// TIA Portal V20 export
FUNCTION "CallManualOperationLines_EM" : Void   // FC66, LAD
// stored: SetENOAutomatically false
   VAR_INPUT
      disableUnit : Bool;
   END_VAR
   VAR_IN_OUT
      manualOperationEm : "LAF_typeManEm";
      manualOperationEmArea : Array[*] of "LAF_typeManOperationArea";
      manualOperationCms : Array[*] of "LAF_typeManOperation";
      Axis : Array[*] of "LBC_typeAxisControlInterface";
      Axis64Pos : Array[*] of "LBC_typeAxis64PosInterface";
      AxisSfotCam : Array[*] of "LER_typeSoftCamRelation";
      Sina : Array[*] of "LBC_typeSinaSpeedInterface";
      twoWayAcutor : Array[*] of "LBC_typeTwoWayActuatorInterface";
      Status : Array[*] of Word;
      errorID : Array[*] of Word;
   END_VAR
   VAR_TEMP
      tempLowerBoundAxis : Int;
      tempUpperBoundAxis : Int;
      tempLowerBoundAxis64Pos : Int;
      tempUpperBoundAxis64Pos : Int;
      tempLowerBoundSina : Int;
      tempUpperBoundSina : Int;
      tempLowerBoundTwoWayAct : Int;
      tempUpperBoundTwoWayAct : Int;
      tempEnd : Bool;
   END_VAR
BEGIN

REGION Network 1: Detect lower and upper bound of the array for further processing
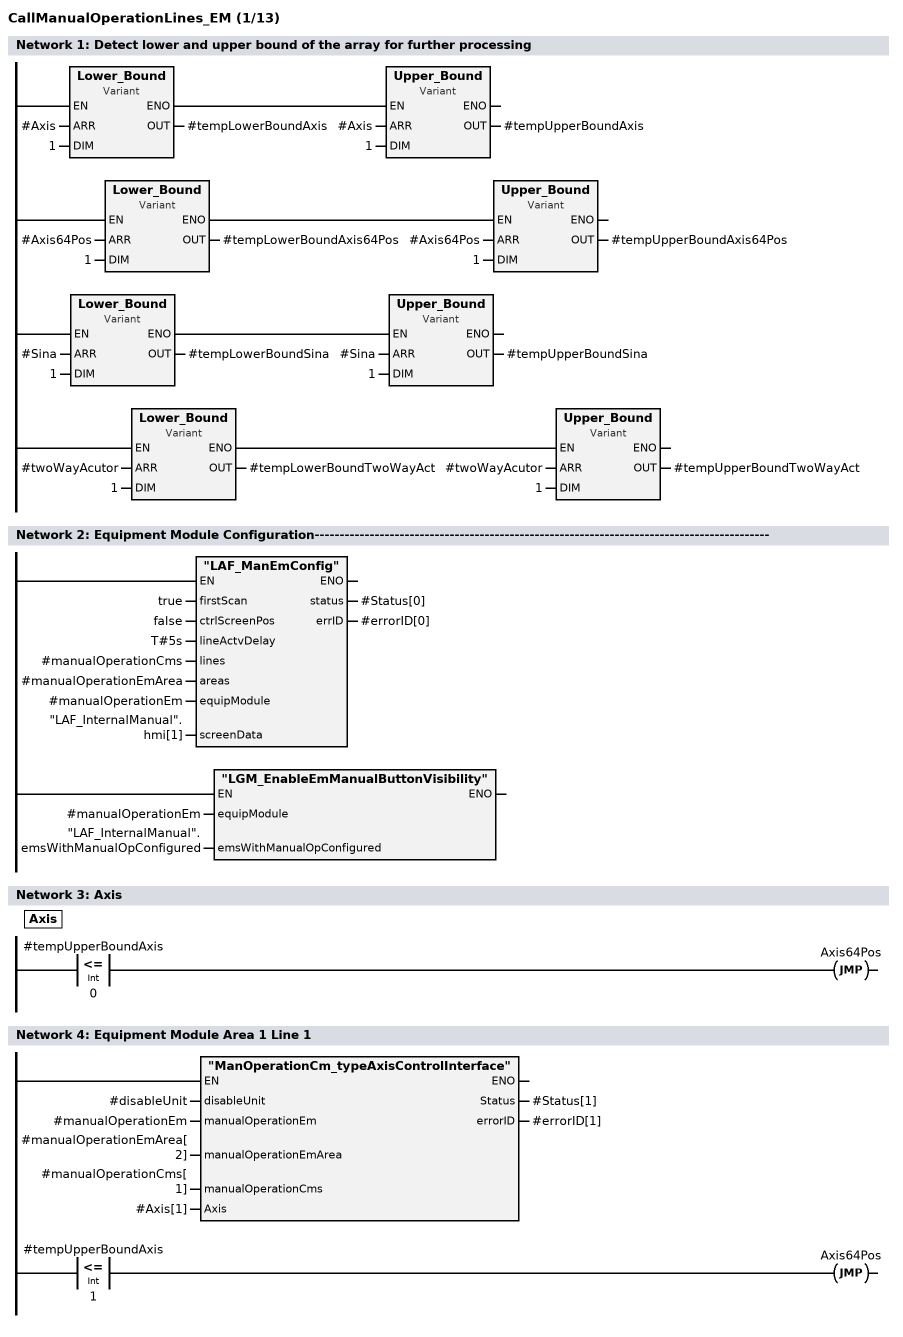
   // no SCL statement known for Lower_Bound, Upper_Bound: written as a call
   // ENO of a box is taken as its EN; it also drops when the box reports an error
   Lower_Bound(arr := #Axis, dim := 1, out => #tempLowerBoundAxis);
   Upper_Bound(arr := #Axis, dim := 1, out => #tempUpperBoundAxis);
   Lower_Bound(arr := #Axis64Pos, dim := 1, out => #tempLowerBoundAxis64Pos);
   Upper_Bound(arr := #Axis64Pos, dim := 1, out => #tempUpperBoundAxis64Pos);
   Lower_Bound(arr := #Sina, dim := 1, out => #tempLowerBoundSina);
   Upper_Bound(arr := #Sina, dim := 1, out => #tempUpperBoundSina);
   Lower_Bound(arr := #twoWayAcutor, dim := 1, out => #tempLowerBoundTwoWayAct);
   Upper_Bound(arr := #twoWayAcutor, dim := 1, out => #tempUpperBoundTwoWayAct);
END_REGION

REGION Network 2: Equipment Module Configuration-------------------------------------------------------------------------------------------
   RUNG wire#powerrail
      "LAF_ManEmConfig"(firstScan := true, ctrlScreenPos := false, lineActvDelay := T#5s, lines := #manualOperationCms, areas := #manualOperationEmArea, equipModule := #manualOperationEm, screenData := "LAF_InternalManual".hmi[1], status => #Status[0], errID => #errorID[0])
   END_RUNG
   RUNG wire#powerrail
      "LGM_EnableEmManualButtonVisibility"(equipModule := #manualOperationEm, emsWithManualOpConfigured := "LAF_InternalManual".emsWithManualOpConfigured)
   END_RUNG
   // the same network as SCL:
   "LAF_ManEmConfig"(firstScan := true,
                     ctrlScreenPos := false,
                     lineActvDelay := T#5s,
                     lines := #manualOperationCms,
                     areas := #manualOperationEmArea,
                     equipModule := #manualOperationEm,
                     screenData := "LAF_InternalManual".hmi[1],
                     status => #Status[0],
                     errID => #errorID[0]);
   "LGM_EnableEmManualButtonVisibility"(equipModule := #manualOperationEm,
                           emsWithManualOpConfigured := "LAF_InternalManual".emsWithManualOpConfigured);
END_REGION

REGION Network 3: Axis
   Label( Axis )
   RUNG wire#powerrail
      { S7_Templates := "SrcType := Int" } LE_Contact(in1 := #tempUpperBoundAxis, in2 := 0)
      JumpCoil( Axis64Pos )
   END_RUNG
   // the same network as SCL:
   Axis:
   IF #tempUpperBoundAxis <= 0 THEN GOTO Axis64Pos; END_IF;
END_REGION

REGION Network 4: Equipment Module Area 1 Line 1
   RUNG wire#powerrail
      "ManOperationCm_typeAxisControlInterface"(disableUnit := #disableUnit, manualOperationEm := #manualOperationEm, manualOperationEmArea := #manualOperationEmArea[2], manualOperationCms := #manualOperationCms[1], Axis := #Axis[1], Status => #Status[1], errorID => #errorID[1])
   END_RUNG
   RUNG wire#powerrail
      { S7_Templates := "SrcType := Int" } LE_Contact(in1 := #tempUpperBoundAxis, in2 := 1)
      JumpCoil( Axis64Pos )
   END_RUNG
   // the same network as SCL:
   "ManOperationCm_typeAxisControlInterface"(disableUnit := #disableUnit,
                           manualOperationEm := #manualOperationEm,
                           manualOperationEmArea := #manualOperationEmArea[2],
                           manualOperationCms := #manualOperationCms[1],
                           Axis := #Axis[1],
                           Status => #Status[1],
                           errorID => #errorID[1]);
   IF #tempUpperBoundAxis <= 1 THEN GOTO Axis64Pos; END_IF;
END_REGION

REGION Network 5: Equipment Module Area 1 Line 2
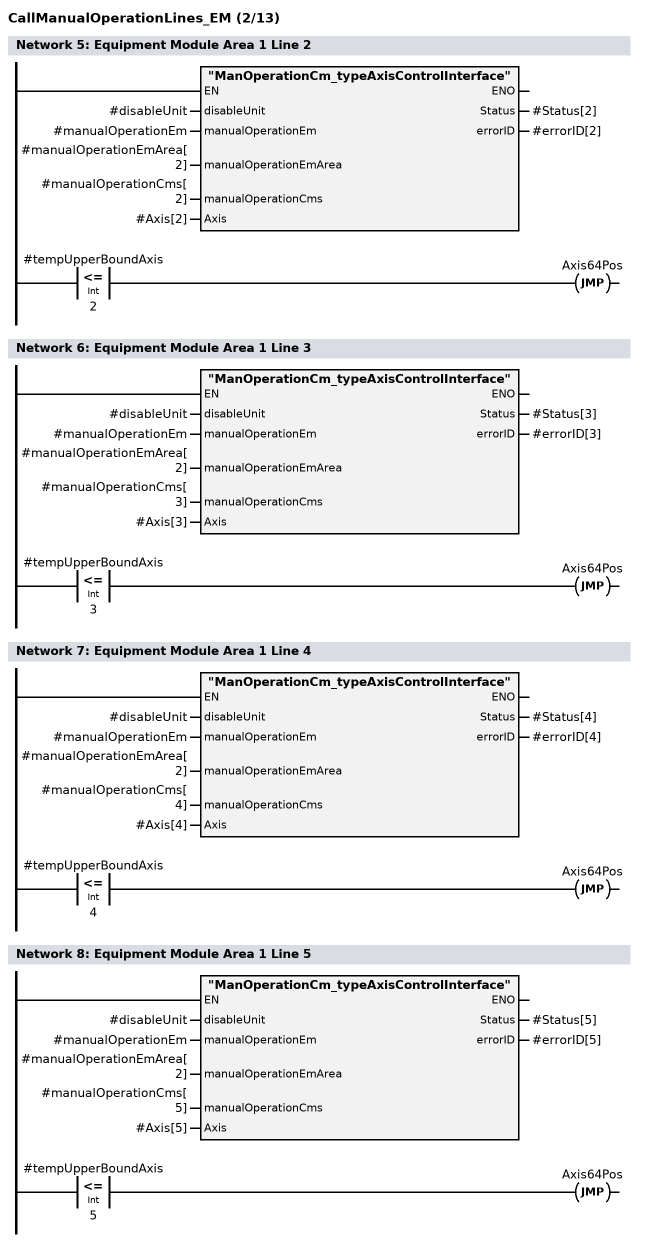
   RUNG wire#powerrail
      "ManOperationCm_typeAxisControlInterface"(disableUnit := #disableUnit, manualOperationEm := #manualOperationEm, manualOperationEmArea := #manualOperationEmArea[2], manualOperationCms := #manualOperationCms[2], Axis := #Axis[2], Status => #Status[2], errorID => #errorID[2])
   END_RUNG
   RUNG wire#powerrail
      { S7_Templates := "SrcType := Int" } LE_Contact(in1 := #tempUpperBoundAxis, in2 := 2)
      JumpCoil( Axis64Pos )
   END_RUNG
   // the same network as SCL:
   "ManOperationCm_typeAxisControlInterface"(disableUnit := #disableUnit,
                           manualOperationEm := #manualOperationEm,
                           manualOperationEmArea := #manualOperationEmArea[2],
                           manualOperationCms := #manualOperationCms[2],
                           Axis := #Axis[2],
                           Status => #Status[2],
                           errorID => #errorID[2]);
   IF #tempUpperBoundAxis <= 2 THEN GOTO Axis64Pos; END_IF;
END_REGION

REGION Network 6: Equipment Module Area 1 Line 3
   RUNG wire#powerrail
      "ManOperationCm_typeAxisControlInterface"(disableUnit := #disableUnit, manualOperationEm := #manualOperationEm, manualOperationEmArea := #manualOperationEmArea[2], manualOperationCms := #manualOperationCms[3], Axis := #Axis[3], Status => #Status[3], errorID => #errorID[3])
   END_RUNG
   RUNG wire#powerrail
      { S7_Templates := "SrcType := Int" } LE_Contact(in1 := #tempUpperBoundAxis, in2 := 3)
      JumpCoil( Axis64Pos )
   END_RUNG
   // the same network as SCL:
   "ManOperationCm_typeAxisControlInterface"(disableUnit := #disableUnit,
                           manualOperationEm := #manualOperationEm,
                           manualOperationEmArea := #manualOperationEmArea[2],
                           manualOperationCms := #manualOperationCms[3],
                           Axis := #Axis[3],
                           Status => #Status[3],
                           errorID => #errorID[3]);
   IF #tempUpperBoundAxis <= 3 THEN GOTO Axis64Pos; END_IF;
END_REGION

REGION Network 7: Equipment Module Area 1 Line 4
   RUNG wire#powerrail
      "ManOperationCm_typeAxisControlInterface"(disableUnit := #disableUnit, manualOperationEm := #manualOperationEm, manualOperationEmArea := #manualOperationEmArea[2], manualOperationCms := #manualOperationCms[4], Axis := #Axis[4], Status => #Status[4], errorID => #errorID[4])
   END_RUNG
   RUNG wire#powerrail
      { S7_Templates := "SrcType := Int" } LE_Contact(in1 := #tempUpperBoundAxis, in2 := 4)
      JumpCoil( Axis64Pos )
   END_RUNG
   // the same network as SCL:
   "ManOperationCm_typeAxisControlInterface"(disableUnit := #disableUnit,
                           manualOperationEm := #manualOperationEm,
                           manualOperationEmArea := #manualOperationEmArea[2],
                           manualOperationCms := #manualOperationCms[4],
                           Axis := #Axis[4],
                           Status => #Status[4],
                           errorID => #errorID[4]);
   IF #tempUpperBoundAxis <= 4 THEN GOTO Axis64Pos; END_IF;
END_REGION

REGION Network 8: Equipment Module Area 1 Line 5
   RUNG wire#powerrail
      "ManOperationCm_typeAxisControlInterface"(disableUnit := #disableUnit, manualOperationEm := #manualOperationEm, manualOperationEmArea := #manualOperationEmArea[2], manualOperationCms := #manualOperationCms[5], Axis := #Axis[5], Status => #Status[5], errorID => #errorID[5])
   END_RUNG
   RUNG wire#powerrail
      { S7_Templates := "SrcType := Int" } LE_Contact(in1 := #tempUpperBoundAxis, in2 := 5)
      JumpCoil( Axis64Pos )
   END_RUNG
   // the same network as SCL:
   "ManOperationCm_typeAxisControlInterface"(disableUnit := #disableUnit,
                           manualOperationEm := #manualOperationEm,
                           manualOperationEmArea := #manualOperationEmArea[2],
                           manualOperationCms := #manualOperationCms[5],
                           Axis := #Axis[5],
                           Status => #Status[5],
                           errorID => #errorID[5]);
   IF #tempUpperBoundAxis <= 5 THEN GOTO Axis64Pos; END_IF;
END_REGION

REGION Network 9: Equipment Module Area 1 Line 6
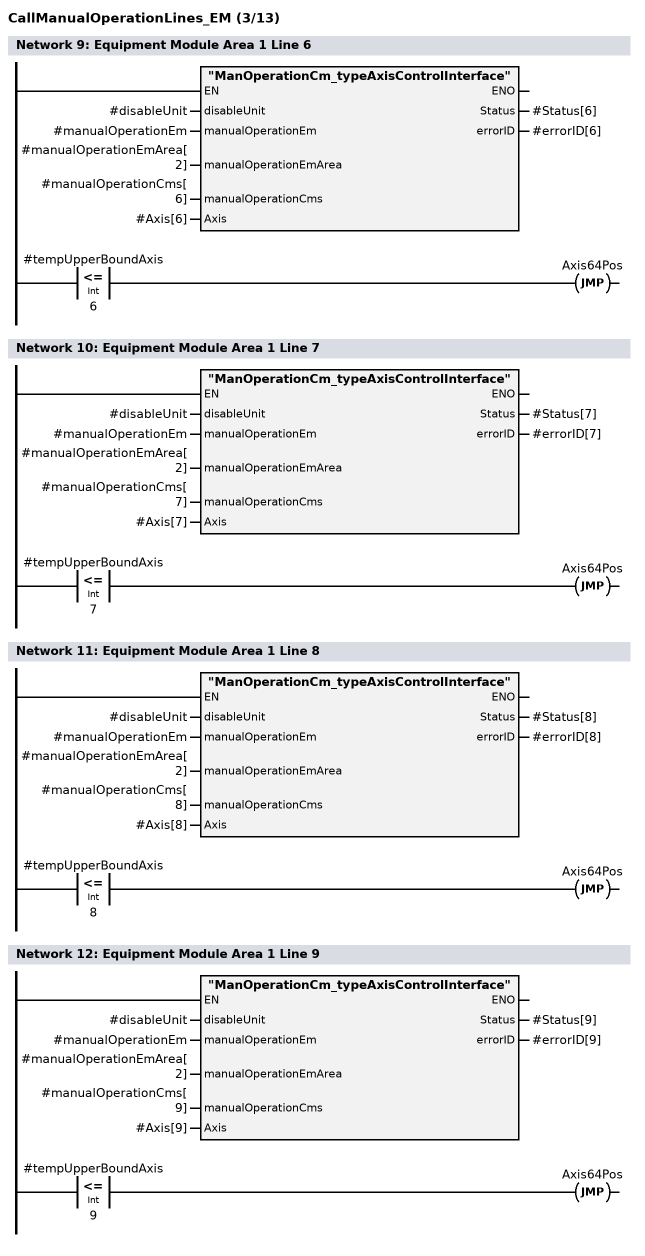
   RUNG wire#powerrail
      "ManOperationCm_typeAxisControlInterface"(disableUnit := #disableUnit, manualOperationEm := #manualOperationEm, manualOperationEmArea := #manualOperationEmArea[2], manualOperationCms := #manualOperationCms[6], Axis := #Axis[6], Status => #Status[6], errorID => #errorID[6])
   END_RUNG
   RUNG wire#powerrail
      { S7_Templates := "SrcType := Int" } LE_Contact(in1 := #tempUpperBoundAxis, in2 := 6)
      JumpCoil( Axis64Pos )
   END_RUNG
   // the same network as SCL:
   "ManOperationCm_typeAxisControlInterface"(disableUnit := #disableUnit,
                           manualOperationEm := #manualOperationEm,
                           manualOperationEmArea := #manualOperationEmArea[2],
                           manualOperationCms := #manualOperationCms[6],
                           Axis := #Axis[6],
                           Status => #Status[6],
                           errorID => #errorID[6]);
   IF #tempUpperBoundAxis <= 6 THEN GOTO Axis64Pos; END_IF;
END_REGION

REGION Network 10: Equipment Module Area 1 Line 7
   RUNG wire#powerrail
      "ManOperationCm_typeAxisControlInterface"(disableUnit := #disableUnit, manualOperationEm := #manualOperationEm, manualOperationEmArea := #manualOperationEmArea[2], manualOperationCms := #manualOperationCms[7], Axis := #Axis[7], Status => #Status[7], errorID => #errorID[7])
   END_RUNG
   RUNG wire#powerrail
      { S7_Templates := "SrcType := Int" } LE_Contact(in1 := #tempUpperBoundAxis, in2 := 7)
      JumpCoil( Axis64Pos )
   END_RUNG
   // the same network as SCL:
   "ManOperationCm_typeAxisControlInterface"(disableUnit := #disableUnit,
                           manualOperationEm := #manualOperationEm,
                           manualOperationEmArea := #manualOperationEmArea[2],
                           manualOperationCms := #manualOperationCms[7],
                           Axis := #Axis[7],
                           Status => #Status[7],
                           errorID => #errorID[7]);
   IF #tempUpperBoundAxis <= 7 THEN GOTO Axis64Pos; END_IF;
END_REGION

REGION Network 11: Equipment Module Area 1 Line 8
   RUNG wire#powerrail
      "ManOperationCm_typeAxisControlInterface"(disableUnit := #disableUnit, manualOperationEm := #manualOperationEm, manualOperationEmArea := #manualOperationEmArea[2], manualOperationCms := #manualOperationCms[8], Axis := #Axis[8], Status => #Status[8], errorID => #errorID[8])
   END_RUNG
   RUNG wire#powerrail
      { S7_Templates := "SrcType := Int" } LE_Contact(in1 := #tempUpperBoundAxis, in2 := 8)
      JumpCoil( Axis64Pos )
   END_RUNG
   // the same network as SCL:
   "ManOperationCm_typeAxisControlInterface"(disableUnit := #disableUnit,
                           manualOperationEm := #manualOperationEm,
                           manualOperationEmArea := #manualOperationEmArea[2],
                           manualOperationCms := #manualOperationCms[8],
                           Axis := #Axis[8],
                           Status => #Status[8],
                           errorID => #errorID[8]);
   IF #tempUpperBoundAxis <= 8 THEN GOTO Axis64Pos; END_IF;
END_REGION

REGION Network 12: Equipment Module Area 1 Line 9
   RUNG wire#powerrail
      "ManOperationCm_typeAxisControlInterface"(disableUnit := #disableUnit, manualOperationEm := #manualOperationEm, manualOperationEmArea := #manualOperationEmArea[2], manualOperationCms := #manualOperationCms[9], Axis := #Axis[9], Status => #Status[9], errorID => #errorID[9])
   END_RUNG
   RUNG wire#powerrail
      { S7_Templates := "SrcType := Int" } LE_Contact(in1 := #tempUpperBoundAxis, in2 := 9)
      JumpCoil( Axis64Pos )
   END_RUNG
   // the same network as SCL:
   "ManOperationCm_typeAxisControlInterface"(disableUnit := #disableUnit,
                           manualOperationEm := #manualOperationEm,
                           manualOperationEmArea := #manualOperationEmArea[2],
                           manualOperationCms := #manualOperationCms[9],
                           Axis := #Axis[9],
                           Status => #Status[9],
                           errorID => #errorID[9]);
   IF #tempUpperBoundAxis <= 9 THEN GOTO Axis64Pos; END_IF;
END_REGION

REGION Network 13: Equipment Module Area 1 Line 10
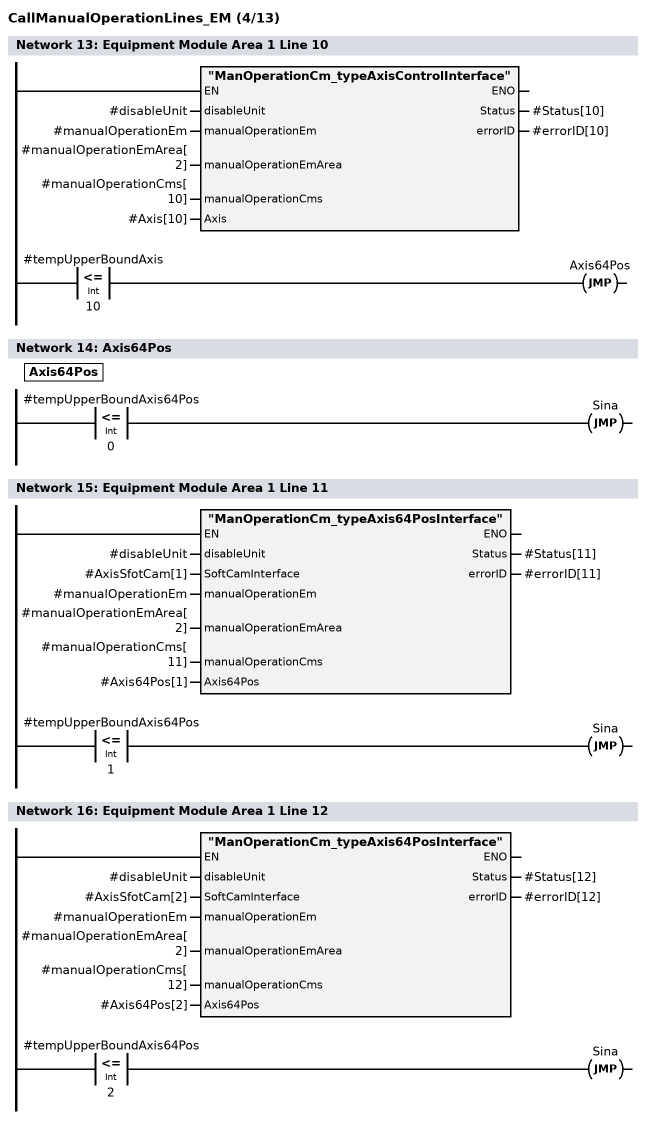
   RUNG wire#powerrail
      "ManOperationCm_typeAxisControlInterface"(disableUnit := #disableUnit, manualOperationEm := #manualOperationEm, manualOperationEmArea := #manualOperationEmArea[2], manualOperationCms := #manualOperationCms[10], Axis := #Axis[10], Status => #Status[10], errorID => #errorID[10])
   END_RUNG
   RUNG wire#powerrail
      { S7_Templates := "SrcType := Int" } LE_Contact(in1 := #tempUpperBoundAxis, in2 := 10)
      JumpCoil( Axis64Pos )
   END_RUNG
   // the same network as SCL:
   "ManOperationCm_typeAxisControlInterface"(disableUnit := #disableUnit,
                           manualOperationEm := #manualOperationEm,
                           manualOperationEmArea := #manualOperationEmArea[2],
                           manualOperationCms := #manualOperationCms[10],
                           Axis := #Axis[10],
                           Status => #Status[10],
                           errorID => #errorID[10]);
   IF #tempUpperBoundAxis <= 10 THEN GOTO Axis64Pos; END_IF;
END_REGION

REGION Network 14: Axis64Pos
   Label( Axis64Pos )
   RUNG wire#powerrail
      { S7_Templates := "SrcType := Int" } LE_Contact(in1 := #tempUpperBoundAxis64Pos, in2 := 0)
      JumpCoil( Sina )
   END_RUNG
   // the same network as SCL:
   Axis64Pos:
   IF #tempUpperBoundAxis64Pos <= 0 THEN GOTO Sina; END_IF;
END_REGION

REGION Network 15: Equipment Module Area 1 Line 11
   RUNG wire#powerrail
      "ManOperationCm_typeAxis64PosInterface"(disableUnit := #disableUnit, SoftCamInterface := #AxisSfotCam[1], manualOperationEm := #manualOperationEm, manualOperationEmArea := #manualOperationEmArea[2], manualOperationCms := #manualOperationCms[11], Axis64Pos := #Axis64Pos[1], Status => #Status[11], errorID => #errorID[11])
   END_RUNG
   RUNG wire#powerrail
      { S7_Templates := "SrcType := Int" } LE_Contact(in1 := #tempUpperBoundAxis64Pos, in2 := 1)
      JumpCoil( Sina )
   END_RUNG
   // the same network as SCL:
   "ManOperationCm_typeAxis64PosInterface"(disableUnit := #disableUnit,
                           SoftCamInterface := #AxisSfotCam[1],
                           manualOperationEm := #manualOperationEm,
                           manualOperationEmArea := #manualOperationEmArea[2],
                           manualOperationCms := #manualOperationCms[11],
                           Axis64Pos := #Axis64Pos[1],
                           Status => #Status[11],
                           errorID => #errorID[11]);
   IF #tempUpperBoundAxis64Pos <= 1 THEN GOTO Sina; END_IF;
END_REGION

REGION Network 16: Equipment Module Area 1 Line 12
   RUNG wire#powerrail
      "ManOperationCm_typeAxis64PosInterface"(disableUnit := #disableUnit, SoftCamInterface := #AxisSfotCam[2], manualOperationEm := #manualOperationEm, manualOperationEmArea := #manualOperationEmArea[2], manualOperationCms := #manualOperationCms[12], Axis64Pos := #Axis64Pos[2], Status => #Status[12], errorID => #errorID[12])
   END_RUNG
   RUNG wire#powerrail
      { S7_Templates := "SrcType := Int" } LE_Contact(in1 := #tempUpperBoundAxis64Pos, in2 := 2)
      JumpCoil( Sina )
   END_RUNG
   // the same network as SCL:
   "ManOperationCm_typeAxis64PosInterface"(disableUnit := #disableUnit,
                           SoftCamInterface := #AxisSfotCam[2],
                           manualOperationEm := #manualOperationEm,
                           manualOperationEmArea := #manualOperationEmArea[2],
                           manualOperationCms := #manualOperationCms[12],
                           Axis64Pos := #Axis64Pos[2],
                           Status => #Status[12],
                           errorID => #errorID[12]);
   IF #tempUpperBoundAxis64Pos <= 2 THEN GOTO Sina; END_IF;
END_REGION

REGION Network 17: Equipment Module Area 1 Line 13
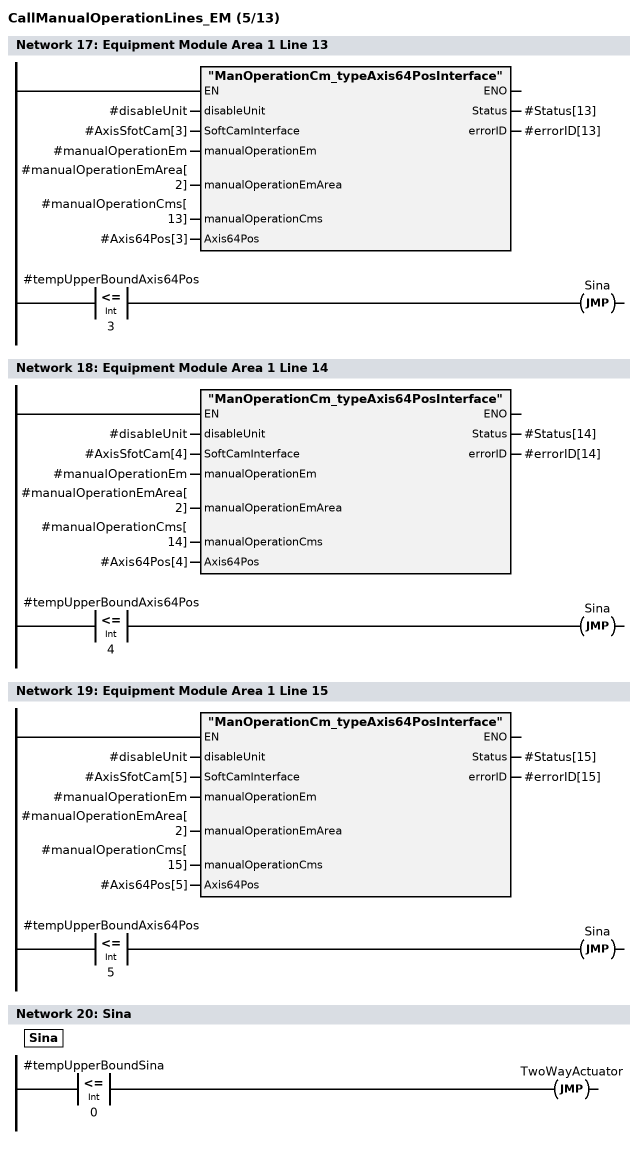
   RUNG wire#powerrail
      "ManOperationCm_typeAxis64PosInterface"(disableUnit := #disableUnit, SoftCamInterface := #AxisSfotCam[3], manualOperationEm := #manualOperationEm, manualOperationEmArea := #manualOperationEmArea[2], manualOperationCms := #manualOperationCms[13], Axis64Pos := #Axis64Pos[3], Status => #Status[13], errorID => #errorID[13])
   END_RUNG
   RUNG wire#powerrail
      { S7_Templates := "SrcType := Int" } LE_Contact(in1 := #tempUpperBoundAxis64Pos, in2 := 3)
      JumpCoil( Sina )
   END_RUNG
   // the same network as SCL:
   "ManOperationCm_typeAxis64PosInterface"(disableUnit := #disableUnit,
                           SoftCamInterface := #AxisSfotCam[3],
                           manualOperationEm := #manualOperationEm,
                           manualOperationEmArea := #manualOperationEmArea[2],
                           manualOperationCms := #manualOperationCms[13],
                           Axis64Pos := #Axis64Pos[3],
                           Status => #Status[13],
                           errorID => #errorID[13]);
   IF #tempUpperBoundAxis64Pos <= 3 THEN GOTO Sina; END_IF;
END_REGION

REGION Network 18: Equipment Module Area 1 Line 14
   RUNG wire#powerrail
      "ManOperationCm_typeAxis64PosInterface"(disableUnit := #disableUnit, SoftCamInterface := #AxisSfotCam[4], manualOperationEm := #manualOperationEm, manualOperationEmArea := #manualOperationEmArea[2], manualOperationCms := #manualOperationCms[14], Axis64Pos := #Axis64Pos[4], Status => #Status[14], errorID => #errorID[14])
   END_RUNG
   RUNG wire#powerrail
      { S7_Templates := "SrcType := Int" } LE_Contact(in1 := #tempUpperBoundAxis64Pos, in2 := 4)
      JumpCoil( Sina )
   END_RUNG
   // the same network as SCL:
   "ManOperationCm_typeAxis64PosInterface"(disableUnit := #disableUnit,
                           SoftCamInterface := #AxisSfotCam[4],
                           manualOperationEm := #manualOperationEm,
                           manualOperationEmArea := #manualOperationEmArea[2],
                           manualOperationCms := #manualOperationCms[14],
                           Axis64Pos := #Axis64Pos[4],
                           Status => #Status[14],
                           errorID => #errorID[14]);
   IF #tempUpperBoundAxis64Pos <= 4 THEN GOTO Sina; END_IF;
END_REGION

REGION Network 19: Equipment Module Area 1 Line 15
   RUNG wire#powerrail
      "ManOperationCm_typeAxis64PosInterface"(disableUnit := #disableUnit, SoftCamInterface := #AxisSfotCam[5], manualOperationEm := #manualOperationEm, manualOperationEmArea := #manualOperationEmArea[2], manualOperationCms := #manualOperationCms[15], Axis64Pos := #Axis64Pos[5], Status => #Status[15], errorID => #errorID[15])
   END_RUNG
   RUNG wire#powerrail
      { S7_Templates := "SrcType := Int" } LE_Contact(in1 := #tempUpperBoundAxis64Pos, in2 := 5)
      JumpCoil( Sina )
   END_RUNG
   // the same network as SCL:
   "ManOperationCm_typeAxis64PosInterface"(disableUnit := #disableUnit,
                           SoftCamInterface := #AxisSfotCam[5],
                           manualOperationEm := #manualOperationEm,
                           manualOperationEmArea := #manualOperationEmArea[2],
                           manualOperationCms := #manualOperationCms[15],
                           Axis64Pos := #Axis64Pos[5],
                           Status => #Status[15],
                           errorID => #errorID[15]);
   IF #tempUpperBoundAxis64Pos <= 5 THEN GOTO Sina; END_IF;
END_REGION

REGION Network 20: Sina
   Label( Sina )
   RUNG wire#powerrail
      { S7_Templates := "SrcType := Int" } LE_Contact(in1 := #tempUpperBoundSina, in2 := 0)
      JumpCoil( TwoWayActuator )
   END_RUNG
   // the same network as SCL:
   Sina:
   IF #tempUpperBoundSina <= 0 THEN GOTO TwoWayActuator; END_IF;
END_REGION

REGION Network 21: Equipment Module Area 1 Line 16
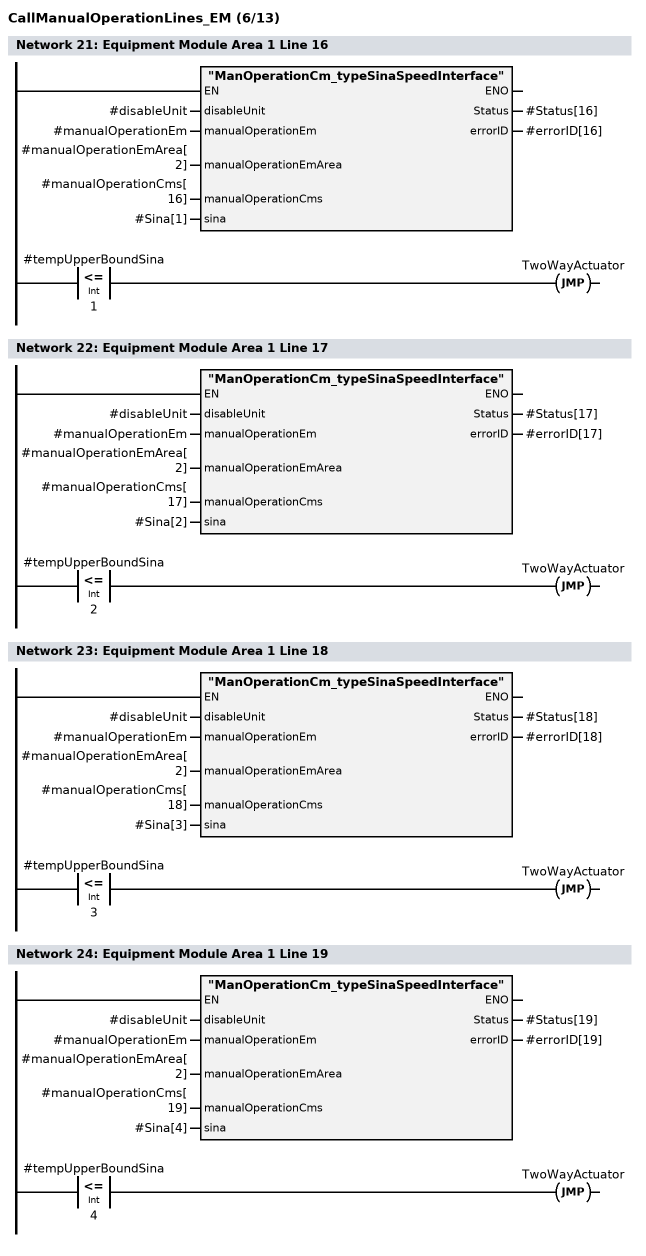
   RUNG wire#powerrail
      "ManOperationCm_typeSinaSpeedInterface"(disableUnit := #disableUnit, manualOperationEm := #manualOperationEm, manualOperationEmArea := #manualOperationEmArea[2], manualOperationCms := #manualOperationCms[16], sina := #Sina[1], Status => #Status[16], errorID => #errorID[16])
   END_RUNG
   RUNG wire#powerrail
      { S7_Templates := "SrcType := Int" } LE_Contact(in1 := #tempUpperBoundSina, in2 := 1)
      JumpCoil( TwoWayActuator )
   END_RUNG
   // the same network as SCL:
   "ManOperationCm_typeSinaSpeedInterface"(disableUnit := #disableUnit,
                           manualOperationEm := #manualOperationEm,
                           manualOperationEmArea := #manualOperationEmArea[2],
                           manualOperationCms := #manualOperationCms[16],
                           sina := #Sina[1],
                           Status => #Status[16],
                           errorID => #errorID[16]);
   IF #tempUpperBoundSina <= 1 THEN GOTO TwoWayActuator; END_IF;
END_REGION

REGION Network 22: Equipment Module Area 1 Line 17
   RUNG wire#powerrail
      "ManOperationCm_typeSinaSpeedInterface"(disableUnit := #disableUnit, manualOperationEm := #manualOperationEm, manualOperationEmArea := #manualOperationEmArea[2], manualOperationCms := #manualOperationCms[17], sina := #Sina[2], Status => #Status[17], errorID => #errorID[17])
   END_RUNG
   RUNG wire#powerrail
      { S7_Templates := "SrcType := Int" } LE_Contact(in1 := #tempUpperBoundSina, in2 := 2)
      JumpCoil( TwoWayActuator )
   END_RUNG
   // the same network as SCL:
   "ManOperationCm_typeSinaSpeedInterface"(disableUnit := #disableUnit,
                           manualOperationEm := #manualOperationEm,
                           manualOperationEmArea := #manualOperationEmArea[2],
                           manualOperationCms := #manualOperationCms[17],
                           sina := #Sina[2],
                           Status => #Status[17],
                           errorID => #errorID[17]);
   IF #tempUpperBoundSina <= 2 THEN GOTO TwoWayActuator; END_IF;
END_REGION

REGION Network 23: Equipment Module Area 1 Line 18
   RUNG wire#powerrail
      "ManOperationCm_typeSinaSpeedInterface"(disableUnit := #disableUnit, manualOperationEm := #manualOperationEm, manualOperationEmArea := #manualOperationEmArea[2], manualOperationCms := #manualOperationCms[18], sina := #Sina[3], Status => #Status[18], errorID => #errorID[18])
   END_RUNG
   RUNG wire#powerrail
      { S7_Templates := "SrcType := Int" } LE_Contact(in1 := #tempUpperBoundSina, in2 := 3)
      JumpCoil( TwoWayActuator )
   END_RUNG
   // the same network as SCL:
   "ManOperationCm_typeSinaSpeedInterface"(disableUnit := #disableUnit,
                           manualOperationEm := #manualOperationEm,
                           manualOperationEmArea := #manualOperationEmArea[2],
                           manualOperationCms := #manualOperationCms[18],
                           sina := #Sina[3],
                           Status => #Status[18],
                           errorID => #errorID[18]);
   IF #tempUpperBoundSina <= 3 THEN GOTO TwoWayActuator; END_IF;
END_REGION

REGION Network 24: Equipment Module Area 1 Line 19
   RUNG wire#powerrail
      "ManOperationCm_typeSinaSpeedInterface"(disableUnit := #disableUnit, manualOperationEm := #manualOperationEm, manualOperationEmArea := #manualOperationEmArea[2], manualOperationCms := #manualOperationCms[19], sina := #Sina[4], Status => #Status[19], errorID => #errorID[19])
   END_RUNG
   RUNG wire#powerrail
      { S7_Templates := "SrcType := Int" } LE_Contact(in1 := #tempUpperBoundSina, in2 := 4)
      JumpCoil( TwoWayActuator )
   END_RUNG
   // the same network as SCL:
   "ManOperationCm_typeSinaSpeedInterface"(disableUnit := #disableUnit,
                           manualOperationEm := #manualOperationEm,
                           manualOperationEmArea := #manualOperationEmArea[2],
                           manualOperationCms := #manualOperationCms[19],
                           sina := #Sina[4],
                           Status => #Status[19],
                           errorID => #errorID[19]);
   IF #tempUpperBoundSina <= 4 THEN GOTO TwoWayActuator; END_IF;
END_REGION

REGION Network 25: Equipment Module Area 1 Line 20
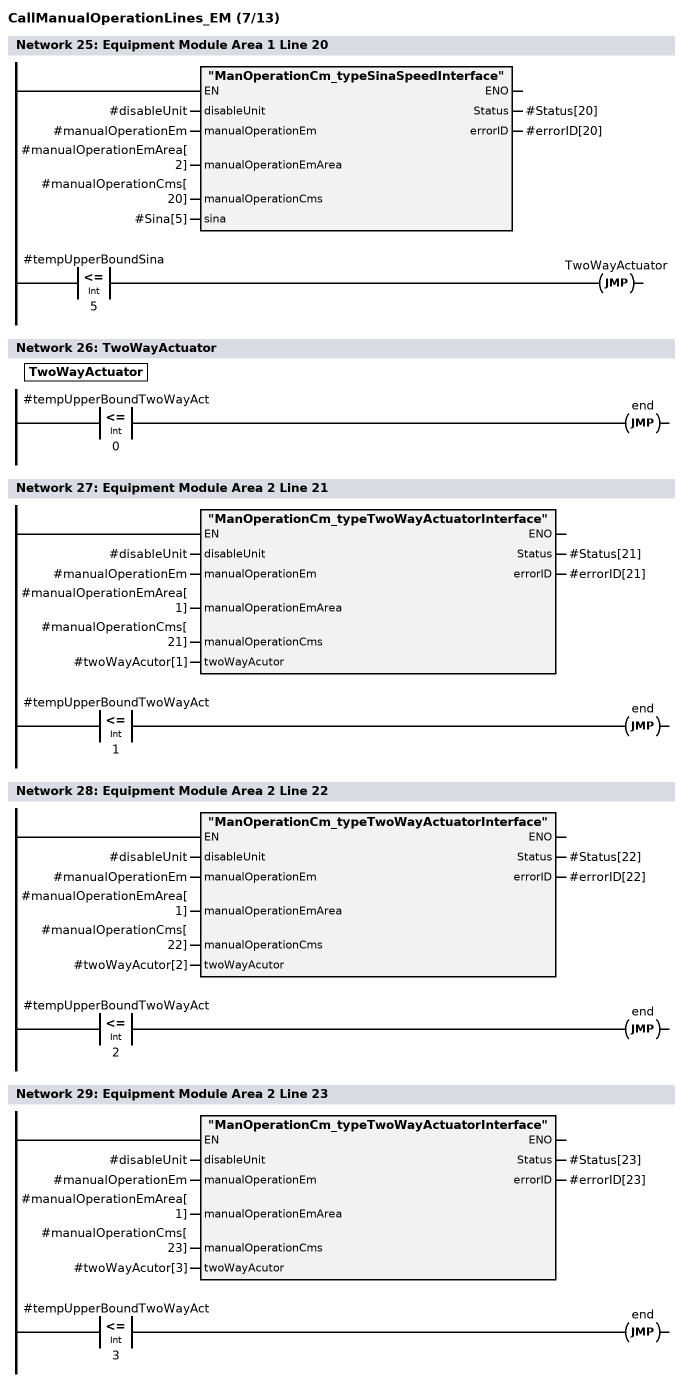
   RUNG wire#powerrail
      "ManOperationCm_typeSinaSpeedInterface"(disableUnit := #disableUnit, manualOperationEm := #manualOperationEm, manualOperationEmArea := #manualOperationEmArea[2], manualOperationCms := #manualOperationCms[20], sina := #Sina[5], Status => #Status[20], errorID => #errorID[20])
   END_RUNG
   RUNG wire#powerrail
      { S7_Templates := "SrcType := Int" } LE_Contact(in1 := #tempUpperBoundSina, in2 := 5)
      JumpCoil( TwoWayActuator )
   END_RUNG
   // the same network as SCL:
   "ManOperationCm_typeSinaSpeedInterface"(disableUnit := #disableUnit,
                           manualOperationEm := #manualOperationEm,
                           manualOperationEmArea := #manualOperationEmArea[2],
                           manualOperationCms := #manualOperationCms[20],
                           sina := #Sina[5],
                           Status => #Status[20],
                           errorID => #errorID[20]);
   IF #tempUpperBoundSina <= 5 THEN GOTO TwoWayActuator; END_IF;
END_REGION

REGION Network 26: TwoWayActuator
   Label( TwoWayActuator )
   RUNG wire#powerrail
      { S7_Templates := "SrcType := Int" } LE_Contact(in1 := #tempUpperBoundTwoWayAct, in2 := 0)
      JumpCoil( end )
   END_RUNG
   // the same network as SCL:
   TwoWayActuator:
   IF #tempUpperBoundTwoWayAct <= 0 THEN GOTO end; END_IF;
END_REGION

REGION Network 27: Equipment Module Area 2 Line 21
   RUNG wire#powerrail
      "ManOperationCm_typeTwoWayActuatorInterface"(disableUnit := #disableUnit, manualOperationEm := #manualOperationEm, manualOperationEmArea := #manualOperationEmArea[1], manualOperationCms := #manualOperationCms[21], twoWayAcutor := #twoWayAcutor[1], Status => #Status[21], errorID => #errorID[21])
   END_RUNG
   RUNG wire#powerrail
      { S7_Templates := "SrcType := Int" } LE_Contact(in1 := #tempUpperBoundTwoWayAct, in2 := 1)
      JumpCoil( end )
   END_RUNG
   // the same network as SCL:
   "ManOperationCm_typeTwoWayActuatorInterface"(disableUnit := #disableUnit,
                           manualOperationEm := #manualOperationEm,
                           manualOperationEmArea := #manualOperationEmArea[1],
                           manualOperationCms := #manualOperationCms[21],
                           twoWayAcutor := #twoWayAcutor[1],
                           Status => #Status[21],
                           errorID => #errorID[21]);
   IF #tempUpperBoundTwoWayAct <= 1 THEN GOTO end; END_IF;
END_REGION

REGION Network 28: Equipment Module Area 2 Line 22
   RUNG wire#powerrail
      "ManOperationCm_typeTwoWayActuatorInterface"(disableUnit := #disableUnit, manualOperationEm := #manualOperationEm, manualOperationEmArea := #manualOperationEmArea[1], manualOperationCms := #manualOperationCms[22], twoWayAcutor := #twoWayAcutor[2], Status => #Status[22], errorID => #errorID[22])
   END_RUNG
   RUNG wire#powerrail
      { S7_Templates := "SrcType := Int" } LE_Contact(in1 := #tempUpperBoundTwoWayAct, in2 := 2)
      JumpCoil( end )
   END_RUNG
   // the same network as SCL:
   "ManOperationCm_typeTwoWayActuatorInterface"(disableUnit := #disableUnit,
                           manualOperationEm := #manualOperationEm,
                           manualOperationEmArea := #manualOperationEmArea[1],
                           manualOperationCms := #manualOperationCms[22],
                           twoWayAcutor := #twoWayAcutor[2],
                           Status => #Status[22],
                           errorID => #errorID[22]);
   IF #tempUpperBoundTwoWayAct <= 2 THEN GOTO end; END_IF;
END_REGION

REGION Network 29: Equipment Module Area 2 Line 23
   RUNG wire#powerrail
      "ManOperationCm_typeTwoWayActuatorInterface"(disableUnit := #disableUnit, manualOperationEm := #manualOperationEm, manualOperationEmArea := #manualOperationEmArea[1], manualOperationCms := #manualOperationCms[23], twoWayAcutor := #twoWayAcutor[3], Status => #Status[23], errorID => #errorID[23])
   END_RUNG
   RUNG wire#powerrail
      { S7_Templates := "SrcType := Int" } LE_Contact(in1 := #tempUpperBoundTwoWayAct, in2 := 3)
      JumpCoil( end )
   END_RUNG
   // the same network as SCL:
   "ManOperationCm_typeTwoWayActuatorInterface"(disableUnit := #disableUnit,
                           manualOperationEm := #manualOperationEm,
                           manualOperationEmArea := #manualOperationEmArea[1],
                           manualOperationCms := #manualOperationCms[23],
                           twoWayAcutor := #twoWayAcutor[3],
                           Status => #Status[23],
                           errorID => #errorID[23]);
   IF #tempUpperBoundTwoWayAct <= 3 THEN GOTO end; END_IF;
END_REGION

REGION Network 30: Equipment Module Area 2 Line 24
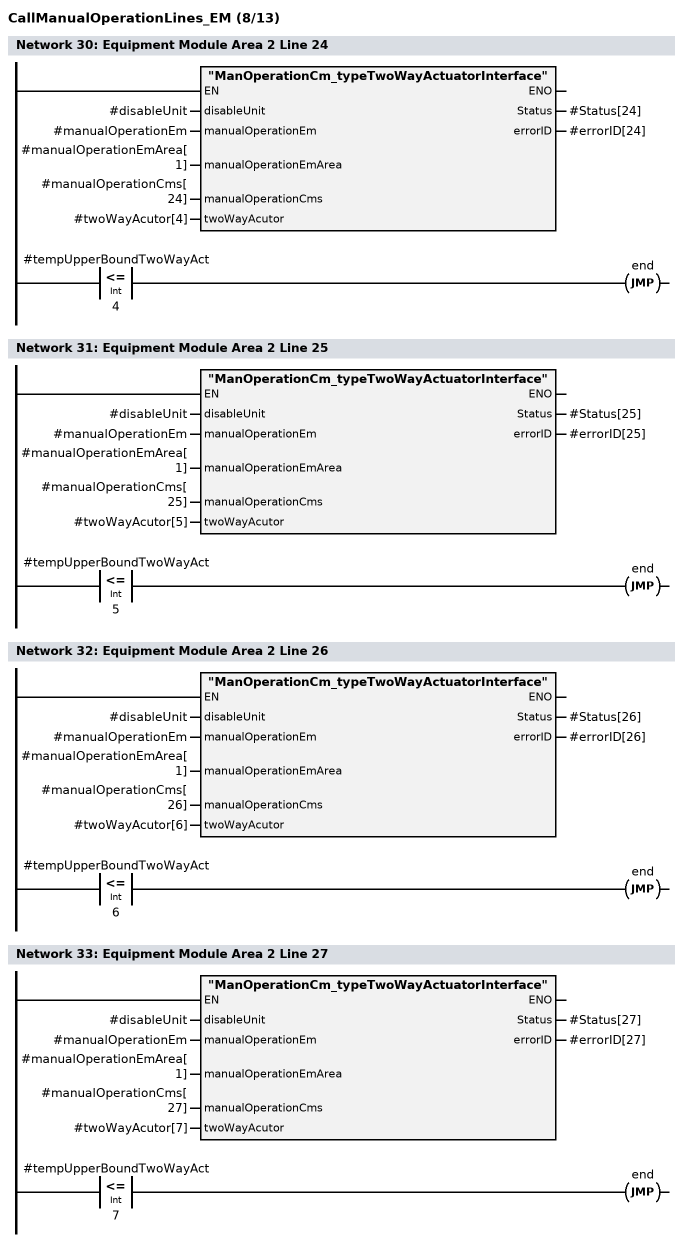
   RUNG wire#powerrail
      "ManOperationCm_typeTwoWayActuatorInterface"(disableUnit := #disableUnit, manualOperationEm := #manualOperationEm, manualOperationEmArea := #manualOperationEmArea[1], manualOperationCms := #manualOperationCms[24], twoWayAcutor := #twoWayAcutor[4], Status => #Status[24], errorID => #errorID[24])
   END_RUNG
   RUNG wire#powerrail
      { S7_Templates := "SrcType := Int" } LE_Contact(in1 := #tempUpperBoundTwoWayAct, in2 := 4)
      JumpCoil( end )
   END_RUNG
   // the same network as SCL:
   "ManOperationCm_typeTwoWayActuatorInterface"(disableUnit := #disableUnit,
                           manualOperationEm := #manualOperationEm,
                           manualOperationEmArea := #manualOperationEmArea[1],
                           manualOperationCms := #manualOperationCms[24],
                           twoWayAcutor := #twoWayAcutor[4],
                           Status => #Status[24],
                           errorID => #errorID[24]);
   IF #tempUpperBoundTwoWayAct <= 4 THEN GOTO end; END_IF;
END_REGION

REGION Network 31: Equipment Module Area 2 Line 25
   RUNG wire#powerrail
      "ManOperationCm_typeTwoWayActuatorInterface"(disableUnit := #disableUnit, manualOperationEm := #manualOperationEm, manualOperationEmArea := #manualOperationEmArea[1], manualOperationCms := #manualOperationCms[25], twoWayAcutor := #twoWayAcutor[5], Status => #Status[25], errorID => #errorID[25])
   END_RUNG
   RUNG wire#powerrail
      { S7_Templates := "SrcType := Int" } LE_Contact(in1 := #tempUpperBoundTwoWayAct, in2 := 5)
      JumpCoil( end )
   END_RUNG
   // the same network as SCL:
   "ManOperationCm_typeTwoWayActuatorInterface"(disableUnit := #disableUnit,
                           manualOperationEm := #manualOperationEm,
                           manualOperationEmArea := #manualOperationEmArea[1],
                           manualOperationCms := #manualOperationCms[25],
                           twoWayAcutor := #twoWayAcutor[5],
                           Status => #Status[25],
                           errorID => #errorID[25]);
   IF #tempUpperBoundTwoWayAct <= 5 THEN GOTO end; END_IF;
END_REGION

REGION Network 32: Equipment Module Area 2 Line 26
   RUNG wire#powerrail
      "ManOperationCm_typeTwoWayActuatorInterface"(disableUnit := #disableUnit, manualOperationEm := #manualOperationEm, manualOperationEmArea := #manualOperationEmArea[1], manualOperationCms := #manualOperationCms[26], twoWayAcutor := #twoWayAcutor[6], Status => #Status[26], errorID => #errorID[26])
   END_RUNG
   RUNG wire#powerrail
      { S7_Templates := "SrcType := Int" } LE_Contact(in1 := #tempUpperBoundTwoWayAct, in2 := 6)
      JumpCoil( end )
   END_RUNG
   // the same network as SCL:
   "ManOperationCm_typeTwoWayActuatorInterface"(disableUnit := #disableUnit,
                           manualOperationEm := #manualOperationEm,
                           manualOperationEmArea := #manualOperationEmArea[1],
                           manualOperationCms := #manualOperationCms[26],
                           twoWayAcutor := #twoWayAcutor[6],
                           Status => #Status[26],
                           errorID => #errorID[26]);
   IF #tempUpperBoundTwoWayAct <= 6 THEN GOTO end; END_IF;
END_REGION

REGION Network 33: Equipment Module Area 2 Line 27
   RUNG wire#powerrail
      "ManOperationCm_typeTwoWayActuatorInterface"(disableUnit := #disableUnit, manualOperationEm := #manualOperationEm, manualOperationEmArea := #manualOperationEmArea[1], manualOperationCms := #manualOperationCms[27], twoWayAcutor := #twoWayAcutor[7], Status => #Status[27], errorID => #errorID[27])
   END_RUNG
   RUNG wire#powerrail
      { S7_Templates := "SrcType := Int" } LE_Contact(in1 := #tempUpperBoundTwoWayAct, in2 := 7)
      JumpCoil( end )
   END_RUNG
   // the same network as SCL:
   "ManOperationCm_typeTwoWayActuatorInterface"(disableUnit := #disableUnit,
                           manualOperationEm := #manualOperationEm,
                           manualOperationEmArea := #manualOperationEmArea[1],
                           manualOperationCms := #manualOperationCms[27],
                           twoWayAcutor := #twoWayAcutor[7],
                           Status => #Status[27],
                           errorID => #errorID[27]);
   IF #tempUpperBoundTwoWayAct <= 7 THEN GOTO end; END_IF;
END_REGION

REGION Network 34: Equipment Module Area 2 Line 28
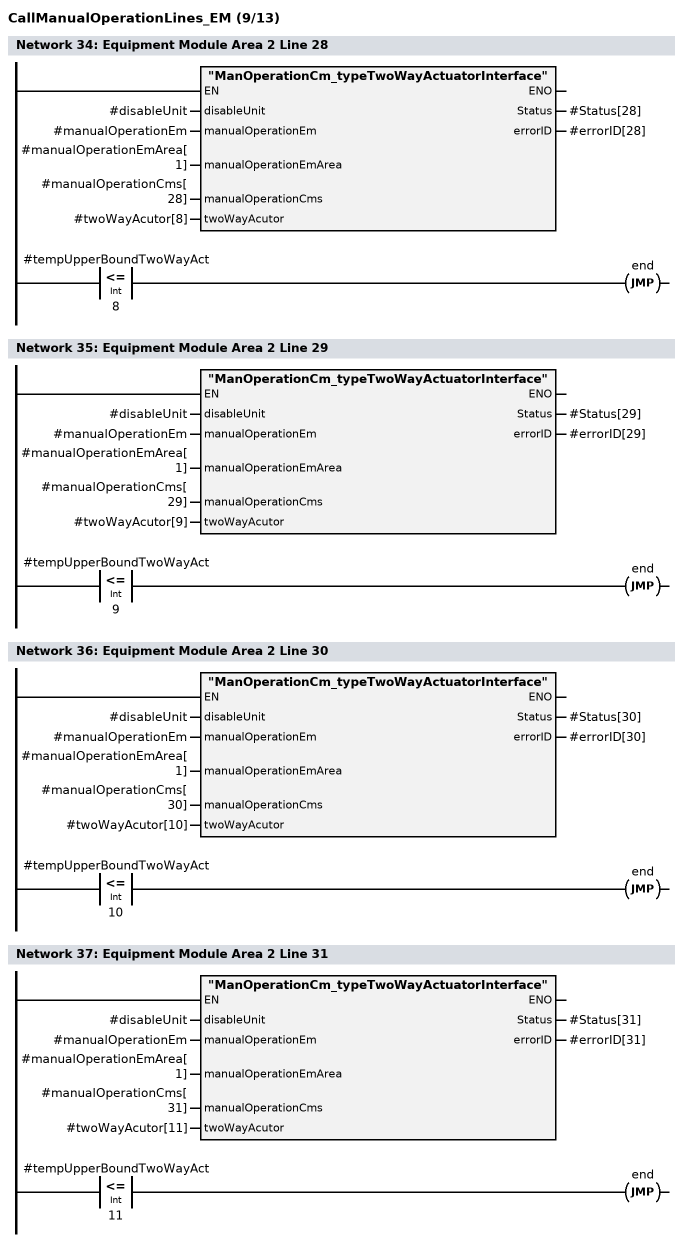
   RUNG wire#powerrail
      "ManOperationCm_typeTwoWayActuatorInterface"(disableUnit := #disableUnit, manualOperationEm := #manualOperationEm, manualOperationEmArea := #manualOperationEmArea[1], manualOperationCms := #manualOperationCms[28], twoWayAcutor := #twoWayAcutor[8], Status => #Status[28], errorID => #errorID[28])
   END_RUNG
   RUNG wire#powerrail
      { S7_Templates := "SrcType := Int" } LE_Contact(in1 := #tempUpperBoundTwoWayAct, in2 := 8)
      JumpCoil( end )
   END_RUNG
   // the same network as SCL:
   "ManOperationCm_typeTwoWayActuatorInterface"(disableUnit := #disableUnit,
                           manualOperationEm := #manualOperationEm,
                           manualOperationEmArea := #manualOperationEmArea[1],
                           manualOperationCms := #manualOperationCms[28],
                           twoWayAcutor := #twoWayAcutor[8],
                           Status => #Status[28],
                           errorID => #errorID[28]);
   IF #tempUpperBoundTwoWayAct <= 8 THEN GOTO end; END_IF;
END_REGION

REGION Network 35: Equipment Module Area 2 Line 29
   RUNG wire#powerrail
      "ManOperationCm_typeTwoWayActuatorInterface"(disableUnit := #disableUnit, manualOperationEm := #manualOperationEm, manualOperationEmArea := #manualOperationEmArea[1], manualOperationCms := #manualOperationCms[29], twoWayAcutor := #twoWayAcutor[9], Status => #Status[29], errorID => #errorID[29])
   END_RUNG
   RUNG wire#powerrail
      { S7_Templates := "SrcType := Int" } LE_Contact(in1 := #tempUpperBoundTwoWayAct, in2 := 9)
      JumpCoil( end )
   END_RUNG
   // the same network as SCL:
   "ManOperationCm_typeTwoWayActuatorInterface"(disableUnit := #disableUnit,
                           manualOperationEm := #manualOperationEm,
                           manualOperationEmArea := #manualOperationEmArea[1],
                           manualOperationCms := #manualOperationCms[29],
                           twoWayAcutor := #twoWayAcutor[9],
                           Status => #Status[29],
                           errorID => #errorID[29]);
   IF #tempUpperBoundTwoWayAct <= 9 THEN GOTO end; END_IF;
END_REGION

REGION Network 36: Equipment Module Area 2 Line 30
   RUNG wire#powerrail
      "ManOperationCm_typeTwoWayActuatorInterface"(disableUnit := #disableUnit, manualOperationEm := #manualOperationEm, manualOperationEmArea := #manualOperationEmArea[1], manualOperationCms := #manualOperationCms[30], twoWayAcutor := #twoWayAcutor[10], Status => #Status[30], errorID => #errorID[30])
   END_RUNG
   RUNG wire#powerrail
      { S7_Templates := "SrcType := Int" } LE_Contact(in1 := #tempUpperBoundTwoWayAct, in2 := 10)
      JumpCoil( end )
   END_RUNG
   // the same network as SCL:
   "ManOperationCm_typeTwoWayActuatorInterface"(disableUnit := #disableUnit,
                           manualOperationEm := #manualOperationEm,
                           manualOperationEmArea := #manualOperationEmArea[1],
                           manualOperationCms := #manualOperationCms[30],
                           twoWayAcutor := #twoWayAcutor[10],
                           Status => #Status[30],
                           errorID => #errorID[30]);
   IF #tempUpperBoundTwoWayAct <= 10 THEN GOTO end; END_IF;
END_REGION

REGION Network 37: Equipment Module Area 2 Line 31
   RUNG wire#powerrail
      "ManOperationCm_typeTwoWayActuatorInterface"(disableUnit := #disableUnit, manualOperationEm := #manualOperationEm, manualOperationEmArea := #manualOperationEmArea[1], manualOperationCms := #manualOperationCms[31], twoWayAcutor := #twoWayAcutor[11], Status => #Status[31], errorID => #errorID[31])
   END_RUNG
   RUNG wire#powerrail
      { S7_Templates := "SrcType := Int" } LE_Contact(in1 := #tempUpperBoundTwoWayAct, in2 := 11)
      JumpCoil( end )
   END_RUNG
   // the same network as SCL:
   "ManOperationCm_typeTwoWayActuatorInterface"(disableUnit := #disableUnit,
                           manualOperationEm := #manualOperationEm,
                           manualOperationEmArea := #manualOperationEmArea[1],
                           manualOperationCms := #manualOperationCms[31],
                           twoWayAcutor := #twoWayAcutor[11],
                           Status => #Status[31],
                           errorID => #errorID[31]);
   IF #tempUpperBoundTwoWayAct <= 11 THEN GOTO end; END_IF;
END_REGION

REGION Network 38: Equipment Module Area 2 Line 32
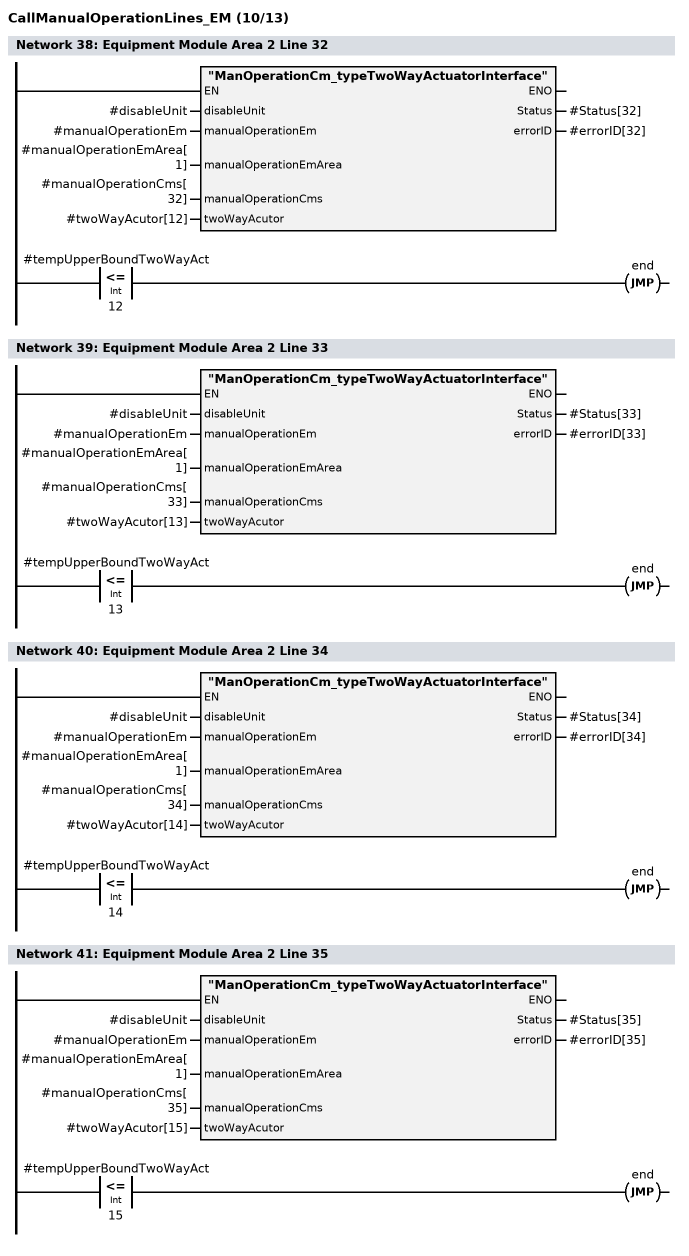
   RUNG wire#powerrail
      "ManOperationCm_typeTwoWayActuatorInterface"(disableUnit := #disableUnit, manualOperationEm := #manualOperationEm, manualOperationEmArea := #manualOperationEmArea[1], manualOperationCms := #manualOperationCms[32], twoWayAcutor := #twoWayAcutor[12], Status => #Status[32], errorID => #errorID[32])
   END_RUNG
   RUNG wire#powerrail
      { S7_Templates := "SrcType := Int" } LE_Contact(in1 := #tempUpperBoundTwoWayAct, in2 := 12)
      JumpCoil( end )
   END_RUNG
   // the same network as SCL:
   "ManOperationCm_typeTwoWayActuatorInterface"(disableUnit := #disableUnit,
                           manualOperationEm := #manualOperationEm,
                           manualOperationEmArea := #manualOperationEmArea[1],
                           manualOperationCms := #manualOperationCms[32],
                           twoWayAcutor := #twoWayAcutor[12],
                           Status => #Status[32],
                           errorID => #errorID[32]);
   IF #tempUpperBoundTwoWayAct <= 12 THEN GOTO end; END_IF;
END_REGION

REGION Network 39: Equipment Module Area 2 Line 33
   RUNG wire#powerrail
      "ManOperationCm_typeTwoWayActuatorInterface"(disableUnit := #disableUnit, manualOperationEm := #manualOperationEm, manualOperationEmArea := #manualOperationEmArea[1], manualOperationCms := #manualOperationCms[33], twoWayAcutor := #twoWayAcutor[13], Status => #Status[33], errorID => #errorID[33])
   END_RUNG
   RUNG wire#powerrail
      { S7_Templates := "SrcType := Int" } LE_Contact(in1 := #tempUpperBoundTwoWayAct, in2 := 13)
      JumpCoil( end )
   END_RUNG
   // the same network as SCL:
   "ManOperationCm_typeTwoWayActuatorInterface"(disableUnit := #disableUnit,
                           manualOperationEm := #manualOperationEm,
                           manualOperationEmArea := #manualOperationEmArea[1],
                           manualOperationCms := #manualOperationCms[33],
                           twoWayAcutor := #twoWayAcutor[13],
                           Status => #Status[33],
                           errorID => #errorID[33]);
   IF #tempUpperBoundTwoWayAct <= 13 THEN GOTO end; END_IF;
END_REGION

REGION Network 40: Equipment Module Area 2 Line 34
   RUNG wire#powerrail
      "ManOperationCm_typeTwoWayActuatorInterface"(disableUnit := #disableUnit, manualOperationEm := #manualOperationEm, manualOperationEmArea := #manualOperationEmArea[1], manualOperationCms := #manualOperationCms[34], twoWayAcutor := #twoWayAcutor[14], Status => #Status[34], errorID => #errorID[34])
   END_RUNG
   RUNG wire#powerrail
      { S7_Templates := "SrcType := Int" } LE_Contact(in1 := #tempUpperBoundTwoWayAct, in2 := 14)
      JumpCoil( end )
   END_RUNG
   // the same network as SCL:
   "ManOperationCm_typeTwoWayActuatorInterface"(disableUnit := #disableUnit,
                           manualOperationEm := #manualOperationEm,
                           manualOperationEmArea := #manualOperationEmArea[1],
                           manualOperationCms := #manualOperationCms[34],
                           twoWayAcutor := #twoWayAcutor[14],
                           Status => #Status[34],
                           errorID => #errorID[34]);
   IF #tempUpperBoundTwoWayAct <= 14 THEN GOTO end; END_IF;
END_REGION

REGION Network 41: Equipment Module Area 2 Line 35
   RUNG wire#powerrail
      "ManOperationCm_typeTwoWayActuatorInterface"(disableUnit := #disableUnit, manualOperationEm := #manualOperationEm, manualOperationEmArea := #manualOperationEmArea[1], manualOperationCms := #manualOperationCms[35], twoWayAcutor := #twoWayAcutor[15], Status => #Status[35], errorID => #errorID[35])
   END_RUNG
   RUNG wire#powerrail
      { S7_Templates := "SrcType := Int" } LE_Contact(in1 := #tempUpperBoundTwoWayAct, in2 := 15)
      JumpCoil( end )
   END_RUNG
   // the same network as SCL:
   "ManOperationCm_typeTwoWayActuatorInterface"(disableUnit := #disableUnit,
                           manualOperationEm := #manualOperationEm,
                           manualOperationEmArea := #manualOperationEmArea[1],
                           manualOperationCms := #manualOperationCms[35],
                           twoWayAcutor := #twoWayAcutor[15],
                           Status => #Status[35],
                           errorID => #errorID[35]);
   IF #tempUpperBoundTwoWayAct <= 15 THEN GOTO end; END_IF;
END_REGION

REGION Network 42: Equipment Module Area 2 Line 36
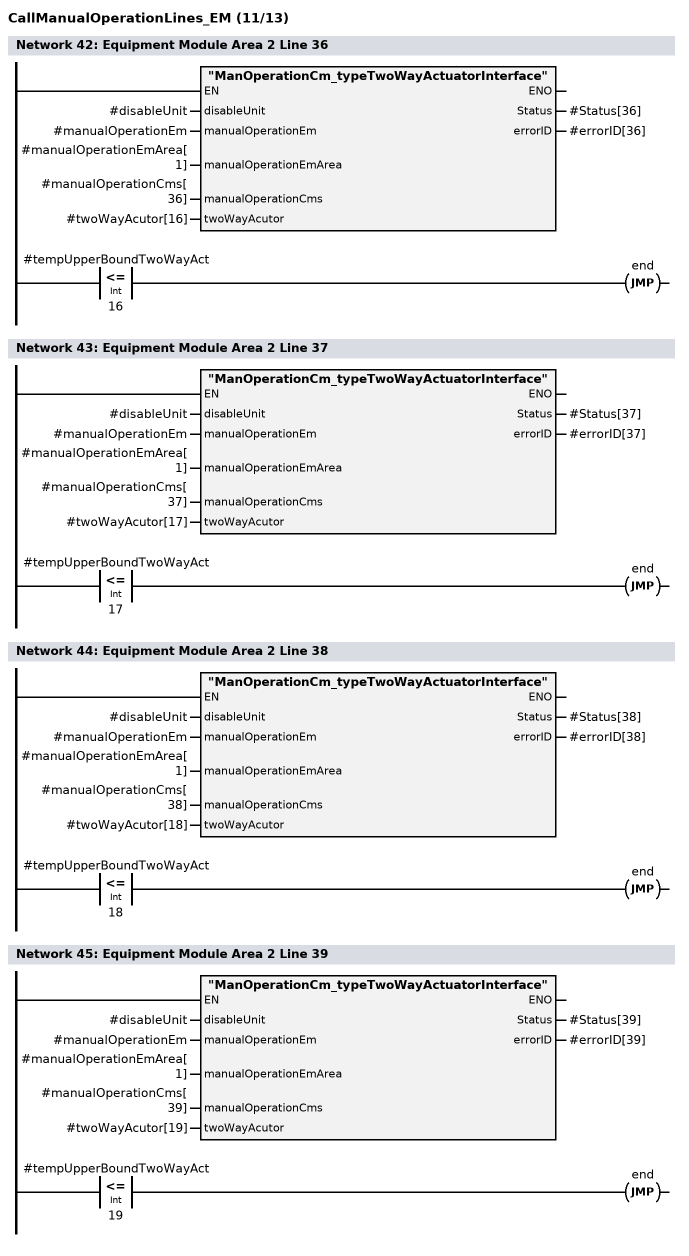
   RUNG wire#powerrail
      "ManOperationCm_typeTwoWayActuatorInterface"(disableUnit := #disableUnit, manualOperationEm := #manualOperationEm, manualOperationEmArea := #manualOperationEmArea[1], manualOperationCms := #manualOperationCms[36], twoWayAcutor := #twoWayAcutor[16], Status => #Status[36], errorID => #errorID[36])
   END_RUNG
   RUNG wire#powerrail
      { S7_Templates := "SrcType := Int" } LE_Contact(in1 := #tempUpperBoundTwoWayAct, in2 := 16)
      JumpCoil( end )
   END_RUNG
   // the same network as SCL:
   "ManOperationCm_typeTwoWayActuatorInterface"(disableUnit := #disableUnit,
                           manualOperationEm := #manualOperationEm,
                           manualOperationEmArea := #manualOperationEmArea[1],
                           manualOperationCms := #manualOperationCms[36],
                           twoWayAcutor := #twoWayAcutor[16],
                           Status => #Status[36],
                           errorID => #errorID[36]);
   IF #tempUpperBoundTwoWayAct <= 16 THEN GOTO end; END_IF;
END_REGION

REGION Network 43: Equipment Module Area 2 Line 37
   RUNG wire#powerrail
      "ManOperationCm_typeTwoWayActuatorInterface"(disableUnit := #disableUnit, manualOperationEm := #manualOperationEm, manualOperationEmArea := #manualOperationEmArea[1], manualOperationCms := #manualOperationCms[37], twoWayAcutor := #twoWayAcutor[17], Status => #Status[37], errorID => #errorID[37])
   END_RUNG
   RUNG wire#powerrail
      { S7_Templates := "SrcType := Int" } LE_Contact(in1 := #tempUpperBoundTwoWayAct, in2 := 17)
      JumpCoil( end )
   END_RUNG
   // the same network as SCL:
   "ManOperationCm_typeTwoWayActuatorInterface"(disableUnit := #disableUnit,
                           manualOperationEm := #manualOperationEm,
                           manualOperationEmArea := #manualOperationEmArea[1],
                           manualOperationCms := #manualOperationCms[37],
                           twoWayAcutor := #twoWayAcutor[17],
                           Status => #Status[37],
                           errorID => #errorID[37]);
   IF #tempUpperBoundTwoWayAct <= 17 THEN GOTO end; END_IF;
END_REGION

REGION Network 44: Equipment Module Area 2 Line 38
   RUNG wire#powerrail
      "ManOperationCm_typeTwoWayActuatorInterface"(disableUnit := #disableUnit, manualOperationEm := #manualOperationEm, manualOperationEmArea := #manualOperationEmArea[1], manualOperationCms := #manualOperationCms[38], twoWayAcutor := #twoWayAcutor[18], Status => #Status[38], errorID => #errorID[38])
   END_RUNG
   RUNG wire#powerrail
      { S7_Templates := "SrcType := Int" } LE_Contact(in1 := #tempUpperBoundTwoWayAct, in2 := 18)
      JumpCoil( end )
   END_RUNG
   // the same network as SCL:
   "ManOperationCm_typeTwoWayActuatorInterface"(disableUnit := #disableUnit,
                           manualOperationEm := #manualOperationEm,
                           manualOperationEmArea := #manualOperationEmArea[1],
                           manualOperationCms := #manualOperationCms[38],
                           twoWayAcutor := #twoWayAcutor[18],
                           Status => #Status[38],
                           errorID => #errorID[38]);
   IF #tempUpperBoundTwoWayAct <= 18 THEN GOTO end; END_IF;
END_REGION

REGION Network 45: Equipment Module Area 2 Line 39
   RUNG wire#powerrail
      "ManOperationCm_typeTwoWayActuatorInterface"(disableUnit := #disableUnit, manualOperationEm := #manualOperationEm, manualOperationEmArea := #manualOperationEmArea[1], manualOperationCms := #manualOperationCms[39], twoWayAcutor := #twoWayAcutor[19], Status => #Status[39], errorID => #errorID[39])
   END_RUNG
   RUNG wire#powerrail
      { S7_Templates := "SrcType := Int" } LE_Contact(in1 := #tempUpperBoundTwoWayAct, in2 := 19)
      JumpCoil( end )
   END_RUNG
   // the same network as SCL:
   "ManOperationCm_typeTwoWayActuatorInterface"(disableUnit := #disableUnit,
                           manualOperationEm := #manualOperationEm,
                           manualOperationEmArea := #manualOperationEmArea[1],
                           manualOperationCms := #manualOperationCms[39],
                           twoWayAcutor := #twoWayAcutor[19],
                           Status => #Status[39],
                           errorID => #errorID[39]);
   IF #tempUpperBoundTwoWayAct <= 19 THEN GOTO end; END_IF;
END_REGION

REGION Network 46: Equipment Module Area 2 Line 40
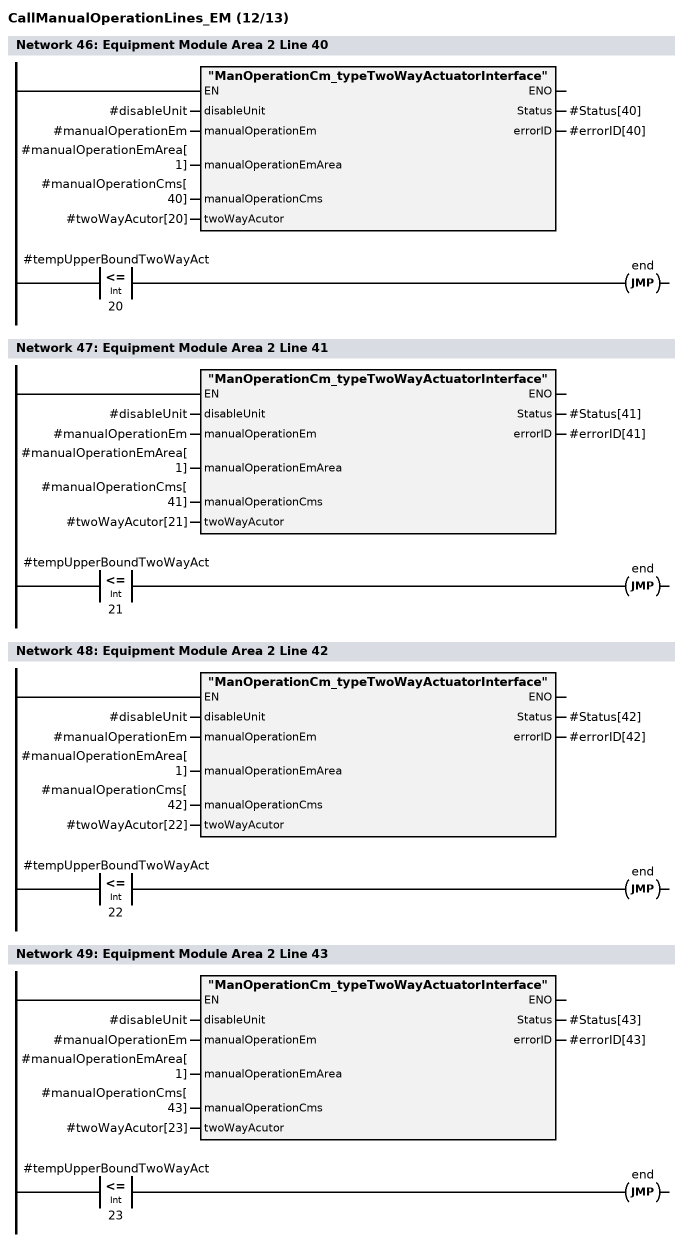
   RUNG wire#powerrail
      "ManOperationCm_typeTwoWayActuatorInterface"(disableUnit := #disableUnit, manualOperationEm := #manualOperationEm, manualOperationEmArea := #manualOperationEmArea[1], manualOperationCms := #manualOperationCms[40], twoWayAcutor := #twoWayAcutor[20], Status => #Status[40], errorID => #errorID[40])
   END_RUNG
   RUNG wire#powerrail
      { S7_Templates := "SrcType := Int" } LE_Contact(in1 := #tempUpperBoundTwoWayAct, in2 := 20)
      JumpCoil( end )
   END_RUNG
   // the same network as SCL:
   "ManOperationCm_typeTwoWayActuatorInterface"(disableUnit := #disableUnit,
                           manualOperationEm := #manualOperationEm,
                           manualOperationEmArea := #manualOperationEmArea[1],
                           manualOperationCms := #manualOperationCms[40],
                           twoWayAcutor := #twoWayAcutor[20],
                           Status => #Status[40],
                           errorID => #errorID[40]);
   IF #tempUpperBoundTwoWayAct <= 20 THEN GOTO end; END_IF;
END_REGION

REGION Network 47: Equipment Module Area 2 Line 41
   RUNG wire#powerrail
      "ManOperationCm_typeTwoWayActuatorInterface"(disableUnit := #disableUnit, manualOperationEm := #manualOperationEm, manualOperationEmArea := #manualOperationEmArea[1], manualOperationCms := #manualOperationCms[41], twoWayAcutor := #twoWayAcutor[21], Status => #Status[41], errorID => #errorID[41])
   END_RUNG
   RUNG wire#powerrail
      { S7_Templates := "SrcType := Int" } LE_Contact(in1 := #tempUpperBoundTwoWayAct, in2 := 21)
      JumpCoil( end )
   END_RUNG
   // the same network as SCL:
   "ManOperationCm_typeTwoWayActuatorInterface"(disableUnit := #disableUnit,
                           manualOperationEm := #manualOperationEm,
                           manualOperationEmArea := #manualOperationEmArea[1],
                           manualOperationCms := #manualOperationCms[41],
                           twoWayAcutor := #twoWayAcutor[21],
                           Status => #Status[41],
                           errorID => #errorID[41]);
   IF #tempUpperBoundTwoWayAct <= 21 THEN GOTO end; END_IF;
END_REGION

REGION Network 48: Equipment Module Area 2 Line 42
   RUNG wire#powerrail
      "ManOperationCm_typeTwoWayActuatorInterface"(disableUnit := #disableUnit, manualOperationEm := #manualOperationEm, manualOperationEmArea := #manualOperationEmArea[1], manualOperationCms := #manualOperationCms[42], twoWayAcutor := #twoWayAcutor[22], Status => #Status[42], errorID => #errorID[42])
   END_RUNG
   RUNG wire#powerrail
      { S7_Templates := "SrcType := Int" } LE_Contact(in1 := #tempUpperBoundTwoWayAct, in2 := 22)
      JumpCoil( end )
   END_RUNG
   // the same network as SCL:
   "ManOperationCm_typeTwoWayActuatorInterface"(disableUnit := #disableUnit,
                           manualOperationEm := #manualOperationEm,
                           manualOperationEmArea := #manualOperationEmArea[1],
                           manualOperationCms := #manualOperationCms[42],
                           twoWayAcutor := #twoWayAcutor[22],
                           Status => #Status[42],
                           errorID => #errorID[42]);
   IF #tempUpperBoundTwoWayAct <= 22 THEN GOTO end; END_IF;
END_REGION

REGION Network 49: Equipment Module Area 2 Line 43
   RUNG wire#powerrail
      "ManOperationCm_typeTwoWayActuatorInterface"(disableUnit := #disableUnit, manualOperationEm := #manualOperationEm, manualOperationEmArea := #manualOperationEmArea[1], manualOperationCms := #manualOperationCms[43], twoWayAcutor := #twoWayAcutor[23], Status => #Status[43], errorID => #errorID[43])
   END_RUNG
   RUNG wire#powerrail
      { S7_Templates := "SrcType := Int" } LE_Contact(in1 := #tempUpperBoundTwoWayAct, in2 := 23)
      JumpCoil( end )
   END_RUNG
   // the same network as SCL:
   "ManOperationCm_typeTwoWayActuatorInterface"(disableUnit := #disableUnit,
                           manualOperationEm := #manualOperationEm,
                           manualOperationEmArea := #manualOperationEmArea[1],
                           manualOperationCms := #manualOperationCms[43],
                           twoWayAcutor := #twoWayAcutor[23],
                           Status => #Status[43],
                           errorID => #errorID[43]);
   IF #tempUpperBoundTwoWayAct <= 23 THEN GOTO end; END_IF;
END_REGION

REGION Network 50: Equipment Module Area 2 Line 44
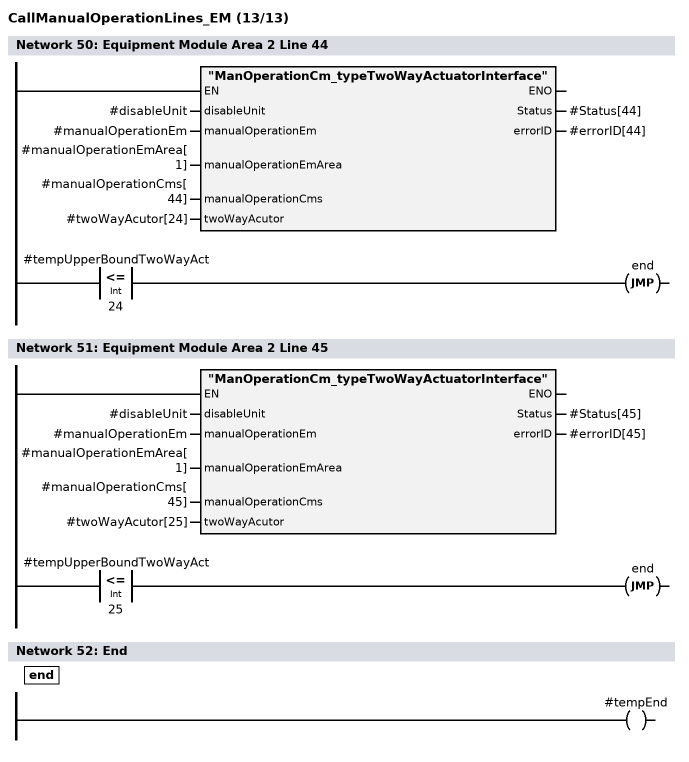
   RUNG wire#powerrail
      "ManOperationCm_typeTwoWayActuatorInterface"(disableUnit := #disableUnit, manualOperationEm := #manualOperationEm, manualOperationEmArea := #manualOperationEmArea[1], manualOperationCms := #manualOperationCms[44], twoWayAcutor := #twoWayAcutor[24], Status => #Status[44], errorID => #errorID[44])
   END_RUNG
   RUNG wire#powerrail
      { S7_Templates := "SrcType := Int" } LE_Contact(in1 := #tempUpperBoundTwoWayAct, in2 := 24)
      JumpCoil( end )
   END_RUNG
   // the same network as SCL:
   "ManOperationCm_typeTwoWayActuatorInterface"(disableUnit := #disableUnit,
                           manualOperationEm := #manualOperationEm,
                           manualOperationEmArea := #manualOperationEmArea[1],
                           manualOperationCms := #manualOperationCms[44],
                           twoWayAcutor := #twoWayAcutor[24],
                           Status => #Status[44],
                           errorID => #errorID[44]);
   IF #tempUpperBoundTwoWayAct <= 24 THEN GOTO end; END_IF;
END_REGION

REGION Network 51: Equipment Module Area 2 Line 45
   RUNG wire#powerrail
      "ManOperationCm_typeTwoWayActuatorInterface"(disableUnit := #disableUnit, manualOperationEm := #manualOperationEm, manualOperationEmArea := #manualOperationEmArea[1], manualOperationCms := #manualOperationCms[45], twoWayAcutor := #twoWayAcutor[25], Status => #Status[45], errorID => #errorID[45])
   END_RUNG
   RUNG wire#powerrail
      { S7_Templates := "SrcType := Int" } LE_Contact(in1 := #tempUpperBoundTwoWayAct, in2 := 25)
      JumpCoil( end )
   END_RUNG
   // the same network as SCL:
   "ManOperationCm_typeTwoWayActuatorInterface"(disableUnit := #disableUnit,
                           manualOperationEm := #manualOperationEm,
                           manualOperationEmArea := #manualOperationEmArea[1],
                           manualOperationCms := #manualOperationCms[45],
                           twoWayAcutor := #twoWayAcutor[25],
                           Status => #Status[45],
                           errorID => #errorID[45]);
   IF #tempUpperBoundTwoWayAct <= 25 THEN GOTO end; END_IF;
END_REGION

REGION Network 52: End
   Label( end )
   RUNG wire#powerrail
      Coil( #tempEnd )
   END_RUNG
   // the same network as SCL:
   end:
   #tempEnd := TRUE;
END_REGION
END_FUNCTION
